(* CoDeSys 2.3.9.41 project: press_4.pro *)
(* Libraries: STANDARD.LIB 4.10.05 11:14:46, IECSFC.LIB 13.4.06 15:51:28, ANALYZATION.LIB 5.10.99 09:05:06, D:\Sespel\Стенды\Пресс\Прорамма\ПЛК100\SysLibTime.lib 17.10.19 08:53:27 *)

(* PLC configuration (modules and I/O channels)
Discrete input 8 bit [ID100] node 0, in %IB0 out %QB0 {Filtrationtime = 10; Filtrationtime = 10; Filtrationtime = 10; Filtrationtime = 10; Filtrationtime = 10; Filtrationtime = 10; Filtrationtime = 10; Filtrationtime = 10; Visibility = No; PinCount = 8; WatchDogPeriod = 1000; PollPeriod = 1}
  AT %IB0.0 [ByteInput] 8 discrete inputs
Discrete output - relay [ID102] node 1, in %IB1 out %QB1 {PinCount = 1; SafeValueBool = FALSE; Visibility = No}
  AT %QX1.0 [BitOutput] relay
Discrete output - relay [ID102] node 2, in %IB2 out %QB2 {PinCount = 1; SafeValueBool = FALSE; Visibility = No}
  AT %QX2.0 [BitOutput] relay
Discrete output - relay [ID102] node 3, in %IB3 out %QB3 {PinCount = 1; SafeValueBool = FALSE; Visibility = No}
  AT %QX3.0 [BitOutput] relay
Discrete output - relay [ID102] node 4, in %IB4 out %QB4 {PinCount = 1; SafeValueBool = FALSE; Visibility = No}
  AT %QX4.0 [BitOutput] relay
Discrete output - relay [ID102] node 5, in %IB5 out %QB5 {PinCount = 1; SafeValueBool = FALSE; Visibility = No}
  AT %QX5.0 [BitOutput] relay
Discrete output - relay [ID102] node 6, in %IB6 out %QB6 {PinCount = 1; SafeValueBool = FALSE; Visibility = No}
  AT %QX6.0 [BitOutput] relay
Special output [ID104] node 7, in %IB7 out %QB7 {Visibility = No; PinCount = 1}
  AT %QX7.0 [BitOutput] Special output
ModBus (Master) [MODBUS_MASTER_ID450] node 8, in %IB8 out %QB8 {Visibility = No}
  AT %QD8.0 [DWordOutput] Last address
  AT %QW8.1 [WordOutput] Last error
  RS-485-1 [COM1_USART] node 0, in %IB8.0 out %QB8.0 {CommunicationSpeed = 57600; Parity = NO PARITY CHECK; BitLength = 8 bits; StopLength = One stop bit; InterfaceType = RS485; FrameOriented = RTU; Timeout = 0; Visibility = No}
AT %QB8.1.0 [ComChannel] Command (0xff - Start)
pr200_dd AT %IW8.1.0.0 [WordInput]
pr200_dd_zad AT %IW8.1.1.0 [WordInput]
pr200_YP AT %IW8.1.2.0 [WordInput]
Cloud [TCP_ID222] node 0, in %IB9.0.0 out %QB9.0.0 {RemotePort = 25502; CloudServerIPFileName = owencloud.txt; CloudToken = MUWOGMWZ; Visibility = No}
cloud_dd AT %QD9.1.0 [FloatOutput]
cloud_YP AT %QW9.2.0 [WordOutput]
cloud_dd_zad AT %QD9.3.0 [FloatOutput]
cloud_zagruzka AT %QD9.4.0 [FloatOutput]
*)

(* POU PLC_PRG, ST *)
PROGRAM PLC_PRG
VAR
	GetTime: CurTimeEx;
	TimeAndDate: SystemTimeDate;
	Sys_Time: SysTime64;
	set_time: BOOL;
	set_date: BOOL;
	MM: UINT;
	SS: UINT;
	HH: UINT;
	D: UINT;
	M: UINT;
	Y: UINT;

	t1:TON;
	t1_trig:R_TRIG;
	t1_in: BOOL;
      t1_real:REAL;
	t1_time:TIME;
	sec: WORD;
	minut:WORD;

	zagruzka_sutki:REAL;
	zagruzka_okrugl:REAL;
END_VAR
cloud_dd:=pr200_dd*0.0084;
cloud_YP:=pr200_YP;
cloud_dd_zad:=pr200_dd_zad*0.1;
cloud_zagruzka:=zagruzka_okrugl;

(*Текущее время*)
TimeAndDate.Day :=0;
TimeAndDate.DayOfWeek :=0;
TimeAndDate.dwHighMsec :=0;
TimeAndDate.dwLowMSecs :=0;
TimeAndDate.Milliseconds :=0;
TimeAndDate.Minute :=0;
TimeAndDate.Second :=0;
TimeAndDate.Hour :=0;
TimeAndDate.Year :=0;
TimeAndDate.Month :=0;
Sys_time.ulHigh :=0;
Sys_time.ulLow :=0;
GetTime (SystemTime:=Sys_Time , TimeDate:= TimeAndDate);

(*Если set_time - истина, то можно менять время*)
IF set_time THEN
	TimeAndDate.Minute:= 48;
	TimeAndDate.Second:=SS;
	TimeAndDate.Hour:=9;
	GetTime (SystemTime:=Sys_Time , TimeDate:= TimeAndDate);
END_IF

(*Обнуляем время по окончанию суток*)
IF TimeAndDate.Hour=0 AND TimeAndDate.Minute =0 AND TimeAndDate.Second =0 THEN
sec:=0;
END_IF

(*Счетчик загруженности за сутки*)
zagruzka_sutki:=sec/864.00;
zagruzka_okrugl:=DINT_TO_REAL(REAL_TO_DINT(zagruzka_sutki*100))/100; (*для огругления до двух знаков после запятой*)

(*Таймер с 1 секундным счетчиком*)
IF pr200_YP=1 THEN
t1_time:=WORD_TO_TIME(1000); (*Преобразовываем значение 1 секунда*)
t1(IN:=t1_in,PT:=t1_time);   (*Запускаем таймер *)
t1_trig(CLK:=t1.Q);
t1_in:=TRUE;
END_IF

IF t1_trig.Q  THEN
sec:=sec+1;
t1_in:=FALSE;
END_IF
END_PROGRAM
